{attribute 'qualified_only'}
{attribute 'strict'}
TYPE ProfileDirectionEnum :
(
	up,
  down
);
END_TYPE

(* stored: Version 1.1.0.1, ProductVersion 3.1.4024.6
   DUT ProfileDirectionEnum: Id {2ff73edb-5bff-447c-9ade-9d123b5bb840} *)
